(* Logix 5000 project; controller blank vendor 1 type 14 code 96 rev 28.11; software revision 28.00 *)

TASK MainTask (continuous, watchdog 500 ms) : MainProgram

MODULES
   Local : vendor 1 type 14 code 96 (ICP 1, rev 28.11)
      relay_output_2 : 1756-IB16 (ICP 2, rev 3.4, Input RPI 20 ms)
      relay_output_4 : 1756-OW16I (ICP 4, rev 3.1, Output RPI 20 ms)
      realy_output_0 : 1756-OW16I (ICP 0, rev 3.1, Output RPI 20 ms)
      relay_output_8 : 1756-IF6I (ICP 8, rev 1.1, Input RPI 100 ms)
      relay_output_7 : vendor 1 type 10 code 4 (ICP 7, rev 1.1, Output RPI 25 ms)
      relay_output_9 : vendor 1 type 12 code 219 (ICP 9, rev 10.1)
END_MODULES

PROGRAM MainProgram   (* main routine MainRoutine *)

ROUTINE MainRoutine   (* ladder *)
END_ROUTINE
END_PROGRAM
